TYPE U_CAM_STATE :
UNION
  stState             : ARRAY[1..MAX_AXIS] OF ST_CAM_STATE;

  byState   AT %Q*    : ARRAY[1..MAX_AXIS] OF
                        ARRAY[1..SIZEOF(ST_CAM_STATE)] OF BYTE;
END_UNION
END_TYPE

(* stored: Version 1.1.0.1, ProductVersion 3.1.4026.13
   DUT U_CAM_STATE: Id {27593e26-7740-4c24-9b35-aa19e32e6825} *)
